// TwinCAT 3 PLC project mobject_graph_plc_pack
// Title: mobject-graph-plc-pack
// Company: mobject
// Author: mobject dev team
// ProjectVersion: 0.19.0
// ProgramVersion: 3.1.4026.22
// libraries:
//   mobject-core,0.10.0,mobject
//   mobject-graph,0.18.0,mobject
//   Tc2_Standard, * (Beckhoff Automation GmbH)
//   Tc2_System, * (Beckhoff Automation GmbH)
//   Tc2_Utilities, * (Beckhoff Automation GmbH)
//   Tc3_Module, * (Beckhoff Automation GmbH)
// project tree:
//   Datatypes/Arrays/ _Array0To7OfByte.TcPOU (not stored)
//   Datatypes/ PlcDatatypePack.TcPOU
//   Datatypes/Structs/ _GUID.TcPOU, _TIMESTRUCT.TcPOU (not stored)
//   Nodes/Converter/DINT_TO_/ Node_DINT_TO_LREAL.TcPOU, Node_DINT_TO_REAL.TcPOU
//   Nodes/Converter/LREAL_TO_/ Node_LREAL_TO_UDINT.TcPOU, Node_LREAL_TO_DINT.TcPOU
//   Nodes/Converter/REAL_TO_/ Node_REAL_TO_UDINT.TcPOU, Node_REAL_TO_DINT.TcPOU
//   Nodes/Converter/UDINT_TO_/ Node_UDINT_TO_REAL.TcPOU, Node_UDINT_TO_LREAL.TcPOU
//   Nodes/Flow/ Node_ForNext.TcPOU, Node_IF.TcPOU, Node_IF_Merge.TcPOU
//   Nodes/Hardware/Digital/ Node_DigitalInput.TcPOU, Node_DigitalOutput.TcPOU
//   Nodes/Logic/ Node_OR.TcPOU, Node_NOT.TcPOU, Node_AND.TcPOU, Node_NOR.TcPOU, Node_NAND.TcPOU, Node_XOR.TcPOU, Node_XNOR.TcPOU
//   Nodes/ PlcNodePack.TcPOU
//   Datatypes/Alias/ _FLOAT.TcPOU (not stored), _HRESULT.TcPOU (not stored)
//   Datatypes/Enums/ _E_TcEventClass.TcPOU (not stored)
//   Nodes/Strings/ Node_CONCAT.TcPOU, Node_DELETE.TcPOU, Node_REPLACE.TcPOU, Node_MID.TcPOU, Node_INSERT.TcPOU, Node_FIND.TcPOU, Node_LEFT.TcPOU, Node_RIGHT.TcPOU, Node_LEN.TcPOU
//   Nodes/TwinCAT/ Node_TwinCATStatus.TcPOU
//   Nodes/Variable/ Node_SetByRef.TcPOU
//   / PlcPack.TcPOU

// ---- Datatypes/PlcDatatypePack.TcPOU
{attribute 'linkalways'} 
{attribute 'no_explicit_call' := 'This FB is a CLASS and must be accessed using methods or properties'}
{attribute 'enable_dynamic_creation'}
FUNCTION_BLOCK PlcDatatypePack
VAR
	
	// alias
    _float : _FLOAT(0.0);
	_hresult : _HRESULT(0);

	// enums
	_e_TcEventClass : _E_TcEventClass(E_TcEventClass.TCEVENTCLASS_NONE);
	
	// structures
	_timestruct : _TIMESTRUCT();
	
END_VAR

METHOD RegisterWithDatatypes
VAR_INPUT
	Datatypes : I_Datatypes;
END_VAR
// alias
Datatypes.RegisterDatatype(_float);
Datatypes.RegisterDatatype(_hresult);

// enums
Datatypes.RegisterDatatype(_e_TcEventClass);

// structures
Datatypes.RegisterDatatype(_timestruct);
END_METHOD

END_FUNCTION_BLOCK

// ---- Datatypes/Structs/_GUID.TcPOU
{attribute 'linkalways'} 
{attribute 'no_explicit_call' := 'This FB is a CLASS and must be accessed using methods or properties'}
{attribute 'enable_dynamic_creation'}
FUNCTION_BLOCK _GUID EXTENDS StructuredDatatypeBase
VAR
	localData : GUID;
	activeData : REFERENCE TO GUID REF= localData;
	_data1 : _DWORD(localData.data1);
	_data2 : _WORD(localData.data2);
    _data3 : _WORD(localData.data3);
	_data4 : _Array0To7OfByte();
END_VAR

PROPERTY PUBLIC Address : PVOID
GET
Address := ADR(activeData);
END_GET
END_PROPERTY

METHOD PUBLIC ClearReference
VAR_INPUT
END_VAR
activeData REF= localData;
SetMemberReference();
END_METHOD

METHOD PUBLIC Clone : I_Datatype
VAR
    pClone : POINTER TO _GUID;
END_VAR
pClone := __NEW(_GUID());
pClone^.Value := Value;
Clone := pClone^;
END_METHOD

PROPERTY PUBLIC Data1 : REFERENCE TO _DWORD
GET
Data1 REF= _data1;
END_GET
END_PROPERTY

PROPERTY PUBLIC Data2 : REFERENCE TO _WORD
GET
Data2 REF= _data2;
END_GET
END_PROPERTY

PROPERTY PUBLIC Data3 : REFERENCE TO _WORD
GET
Data3 REF= _data3;
END_GET
END_PROPERTY

PROPERTY PUBLIC Data4 : REFERENCE TO _Array0To7OfByte
GET
Data4 REF= _data4;
END_GET
END_PROPERTY

METHOD PUBLIC EqualsGuid : BOOL
VAR_INPUT
	guid : GUID;
END_VAR
EqualsGuid := GuidsEqual(adr(guid), this^.Address);
END_METHOD

METHOD FB_init : BOOL
VAR_INPUT
	bInitRetains : BOOL; // if TRUE, the retain variables are initialized (warm start / cold start)
	bInCopyCode : BOOL;  // if TRUE, the instance afterwards gets moved into the copy code (online change)
END_VAR
SetMemberReference();
AddMember('Data1',_data1);
AddMember('Data2',_data2);
AddMember('Data3',_data3);
AddMember('Data4',_data4);
END_METHOD

PROPERTY PUBLIC Identifier : T_MAXSTRING
GET
Identifier := 'GUID';
END_GET
END_PROPERTY

METHOD PROTECTED IsValidGuidString : BOOL
VAR_INPUT
	GuidAsString : STRING;
END_VAR
VAR
	position : INT;
	stringIndex : INT;
	dashCount : INT := 0;
END_VAR
VAR CONSTANT
	CHARACTER_HYPHEN : BYTE := 16#2D;
	CHARACTER_0 : BYTE := 16#30;
	CHARACTER_9 : BYTE := 16#39;
	CHARACTER_A : BYTE := 16#41;
	CHARACTER_F : BYTE := 16#46;
	CHARACTER_LCASE_A : BYTE := 16#61;
	CHARACTER_LCASE_F : BYTE := 16#66;
END_VAR
// Check the overall length of the string (36 including 4 dashes)
IF LEN(GuidAsString) <> 36 THEN
	RETURN;
END_IF

// Check each character
FOR position := 1 TO 36 DO
	stringIndex := position - 1; 
	CASE position OF
		9, 14, 19, 24:
			// Dashes should be at positions 9, 14, 19, 24
			IF GuidAsString[stringIndex] <> CHARACTER_HYPHEN THEN
				RETURN;
			ELSE
				dashCount := dashCount + 1;
			END_IF
		ELSE
			// All other positions should contain hex digits (0-9, A-F, a-f)
			IF NOT ((GuidAsString[stringIndex] >= CHARACTER_0 AND GuidAsString[stringIndex] <= CHARACTER_9) OR 
				(GuidAsString[stringIndex] >= CHARACTER_A AND GuidAsString[stringIndex] <= CHARACTER_F) OR 
				(GuidAsString[stringIndex] >= CHARACTER_LCASE_A AND GuidAsString[stringIndex] <= CHARACTER_LCASE_F)) THEN
				RETURN;
			END_IF
	END_CASE
END_FOR

// Ensure exactly four dashes are present
IF dashCount = 4 THEN
	IsValidGuidString := TRUE;
END_IF
END_METHOD

METHOD PUBLIC MakeReferenceTo
VAR_INPUT
	ReferenceTarget : REFERENCE TO GUID;
END_VAR
activeData REF= ReferenceTarget;
SetMemberReference();
END_METHOD

METHOD PROTECTED SetMemberReference
VAR_INPUT
END_VAR
_data1.MakeReferenceTo(activeData.Data1);
_data2.MakeReferenceTo(activeData.Data2);
_data3.MakeReferenceTo(activeData.Data3);
_data4.MakeReferenceTo(activeData.Data4);
END_METHOD

PROPERTY PUBLIC Size : UDINT
GET
Size := SIZEOF(activeData);
END_GET
END_PROPERTY

METHOD PUBLIC ToString : T_MAXSTRING
VAR_INPUT
END_VAR
ToString := GUID_TO_STRING(activeData);
END_METHOD

METHOD TryDeserializeFrom : BOOL
VAR_INPUT
	Deserializer : I_Deserializer;
	Feedback : I_DeserializerFeedback;
END_VAR
VAR
	localFeedback : DeserializerFeedback;
	guidAsString : T_MAXSTRING;
END_VAR
// this customized version of TryDeserializeFrom allows for the use of string guids. 
// if a string is not found, then it will try to deserialize from an object.
IF Deserializer.TryGetString(guidAsString, localFeedback) THEN	
	IF TryFromString(guidAsString) THEN
		TryDeserializeFrom := TRUE;
		RETURN;
	END_IF
	
	Feedback.LogDeserializationFailedError('Invalid GUID String');	
	RETURN;
END_IF

TryDeserializeFrom := SUPER^.TryDeserializeFrom(Deserializer, Feedback);
END_METHOD

METHOD PUBLIC TryFromString : BOOL;
VAR_INPUT
	GuidAsString : T_MAXSTRING;
END_VAR
IF NOT IsValidGuidString(GuidAsString) THEN
	RETURN;
END_IF

activeData := STRING_TO_GUID(GuidAsString);
TryFromString := true;
END_METHOD

METHOD TryMakeReferenceTo : BOOL
VAR_INPUT
	Target : I_Datatype;
END_VAR
VAR
	pTargetData : POINTER TO GUID;
END_VAR
IF NOT IsEquivalentTo(Target) THEN
	RETURN;
END_IF

pTargetData := Target.Address;
activeData REF= pTargetData^;
SetMemberReference();
TryMakeReferenceTo := TRUE;
END_METHOD

PROPERTY PUBLIC Value : REFERENCE TO GUID
GET
Value REF= activeData;
END_GET
END_PROPERTY

END_FUNCTION_BLOCK

// ---- Nodes/Converter/DINT_TO_/Node_DINT_TO_LREAL.TcPOU
{attribute 'linkalways'} 
{attribute 'no_explicit_call' := 'This FB is a CLASS and must be accessed using methods or properties'}
{attribute 'enable_dynamic_creation'}
FUNCTION_BLOCK FINAL Node_DINT_TO_LREAL EXTENDS Node
VAR
	in : _DINT(0);
	out : _LREAL(0.0);
	success : _BOOL(FALSE);
END_VAR

METHOD PUBLIC  Clone : I_Node
VAR
	pNode : POINTER TO Node_DINT_TO_LREAL;
END_VAR
pNode := __NEW(Node_DINT_TO_LREAL);
Clone := pNode^;
END_METHOD

METHOD FB_init : BOOL
VAR_INPUT
	bInitRetains : BOOL; // if TRUE, the retain variables are initialized (warm start / cold start)
	bInCopyCode : BOOL;  // if TRUE, the instance afterwards gets moved into the copy code (online change)
END_VAR
AddParameter('in', in);
AddOutput('out', out);
AddOutput('success', success);

this^.Metadatum.AddBoolAsMetadata('deprecated', true);
END_METHOD

METHOD PROTECTED OnExecute
VAR
END_VAR
success.Value := TryConvert_DINT_TO_LREAL(in.Value, out.Value);
END_METHOD

END_FUNCTION_BLOCK

// ---- Nodes/Converter/DINT_TO_/Node_DINT_TO_REAL.TcPOU
{attribute 'linkalways'} 
{attribute 'no_explicit_call' := 'This FB is a CLASS and must be accessed using methods or properties'}
{attribute 'enable_dynamic_creation'}
FUNCTION_BLOCK FINAL Node_DINT_TO_REAL EXTENDS Node
VAR
	in : _DINT(0);
	out : _REAL(0.0);
	success : _BOOL(FALSE);
END_VAR

METHOD PUBLIC  Clone : I_Node
VAR
	pNode : POINTER TO Node_DINT_TO_REAL;
END_VAR
pNode := __NEW(Node_DINT_TO_REAL);
Clone := pNode^;
END_METHOD

METHOD FB_init : BOOL
VAR_INPUT
	bInitRetains : BOOL; // if TRUE, the retain variables are initialized (warm start / cold start)
	bInCopyCode : BOOL;  // if TRUE, the instance afterwards gets moved into the copy code (online change)
END_VAR
AddParameter('in', in);
AddOutput('out', out);
AddOutput('success', success);

this^.Metadatum.AddBoolAsMetadata('deprecated', true);
END_METHOD

METHOD PROTECTED OnExecute
VAR
END_VAR
success.Value := TryConvert_DINT_TO_REAL(in.Value, out.Value);
END_METHOD

END_FUNCTION_BLOCK

// ---- Nodes/Converter/LREAL_TO_/Node_LREAL_TO_UDINT.TcPOU
{attribute 'linkalways'} 
{attribute 'no_explicit_call' := 'This FB is a CLASS and must be accessed using methods or properties'}
{attribute 'enable_dynamic_creation'}
FUNCTION_BLOCK FINAL Node_LREAL_TO_UDINT EXTENDS Node
VAR
	in : _LREAL(0.0);
	out : _UDINT(0);
	success : _BOOL(FALSE);
END_VAR

METHOD PUBLIC  Clone : I_Node
VAR
	pNode : POINTER TO Node_LREAL_TO_UDINT;
END_VAR
pNode := __NEW(Node_LREAL_TO_UDINT);
Clone := pNode^;
END_METHOD

METHOD FB_init : BOOL
VAR_INPUT
	bInitRetains : BOOL; // if TRUE, the retain variables are initialized (warm start / cold start)
	bInCopyCode : BOOL;  // if TRUE, the instance afterwards gets moved into the copy code (online change)
END_VAR
AddParameter('in', in);
AddOutput('out', out);
AddOutput('success', success);

this^.Metadatum.AddBoolAsMetadata('deprecated', true);
END_METHOD

METHOD PROTECTED OnExecute
VAR
END_VAR
success.Value := TryConvert_LREAL_TO_UDINT(in.Value, out.Value);
END_METHOD

END_FUNCTION_BLOCK

// ---- Nodes/Converter/LREAL_TO_/Node_LREAL_TO_DINT.TcPOU
{attribute 'linkalways'} 
{attribute 'no_explicit_call' := 'This FB is a CLASS and must be accessed using methods or properties'}
{attribute 'enable_dynamic_creation'}
FUNCTION_BLOCK FINAL Node_LREAL_TO_DINT EXTENDS Node
VAR
	in : _LREAL(0.0);
	out : _DINT(0);
	success : _BOOL(FALSE);
END_VAR

METHOD PUBLIC  Clone : I_Node
VAR
	pNode : POINTER TO Node_LREAL_TO_DINT;
END_VAR
pNode := __NEW(Node_LREAL_TO_DINT);
Clone := pNode^;
END_METHOD

METHOD FB_init : BOOL
VAR_INPUT
	bInitRetains : BOOL; // if TRUE, the retain variables are initialized (warm start / cold start)
	bInCopyCode : BOOL;  // if TRUE, the instance afterwards gets moved into the copy code (online change)
END_VAR
AddParameter('in', in);
AddOutput('out', out);
AddOutput('success', success);

this^.Metadatum.AddBoolAsMetadata('deprecated', true);
END_METHOD

METHOD PROTECTED OnExecute
VAR
END_VAR
success.Value := TryConvert_LREAL_TO_DINT(in.Value, out.Value);
END_METHOD

END_FUNCTION_BLOCK

// ---- Nodes/Converter/REAL_TO_/Node_REAL_TO_UDINT.TcPOU
{attribute 'linkalways'} 
{attribute 'no_explicit_call' := 'This FB is a CLASS and must be accessed using methods or properties'}
{attribute 'enable_dynamic_creation'}
FUNCTION_BLOCK FINAL Node_REAL_TO_UDINT EXTENDS Node
VAR
	in : _REAL(0.0);
	out : _UDINT(0);
	success : _BOOL(FALSE);
END_VAR

METHOD PUBLIC  Clone : I_Node
VAR
	pNode : POINTER TO Node_REAL_TO_UDINT;
END_VAR
pNode := __NEW(Node_REAL_TO_UDINT);
Clone := pNode^;
END_METHOD

METHOD FB_init : BOOL
VAR_INPUT
	bInitRetains : BOOL; // if TRUE, the retain variables are initialized (warm start / cold start)
	bInCopyCode : BOOL;  // if TRUE, the instance afterwards gets moved into the copy code (online change)
END_VAR
AddParameter('in', in);
AddOutput('out', out);
AddOutput('success', success);

this^.Metadatum.AddBoolAsMetadata('deprecated', true);
END_METHOD

METHOD PROTECTED OnExecute
VAR
END_VAR
success.Value := TryConvert_REAL_TO_UDINT(in.Value, out.Value);
END_METHOD

END_FUNCTION_BLOCK

// ---- Nodes/Converter/REAL_TO_/Node_REAL_TO_DINT.TcPOU
{attribute 'linkalways'} 
{attribute 'no_explicit_call' := 'This FB is a CLASS and must be accessed using methods or properties'}
{attribute 'enable_dynamic_creation'}
FUNCTION_BLOCK FINAL Node_REAL_TO_DINT EXTENDS Node
VAR
	in : _REAL(0.0);
	out : _DINT(0);
	success : _BOOL(FALSE);
END_VAR

METHOD PUBLIC  Clone : I_Node
VAR
	pNode : POINTER TO Node_REAL_TO_DINT;
END_VAR
pNode := __NEW(Node_REAL_TO_DINT);
Clone := pNode^;
END_METHOD

METHOD FB_init : BOOL
VAR_INPUT
	bInitRetains : BOOL; // if TRUE, the retain variables are initialized (warm start / cold start)
	bInCopyCode : BOOL;  // if TRUE, the instance afterwards gets moved into the copy code (online change)
END_VAR
AddParameter('in', in);
AddOutput('out', out);
AddOutput('success', success);

this^.Metadatum.AddBoolAsMetadata('deprecated', true);
END_METHOD

METHOD PROTECTED OnExecute
VAR
END_VAR
success.Value := TryConvert_REAL_TO_DINT(in.Value, out.Value);
END_METHOD

END_FUNCTION_BLOCK

// ---- Nodes/Converter/UDINT_TO_/Node_UDINT_TO_REAL.TcPOU
{attribute 'linkalways'} 
{attribute 'no_explicit_call' := 'This FB is a CLASS and must be accessed using methods or properties'}
{attribute 'enable_dynamic_creation'}
FUNCTION_BLOCK FINAL Node_UDINT_TO_REAL EXTENDS Node
VAR
	in : _UDINT(0);
	out : _REAL(0.0);
	success : _BOOL(FALSE);
END_VAR

METHOD PUBLIC  Clone : I_Node
VAR
	pNode : POINTER TO Node_UDINT_TO_REAL;
END_VAR
pNode := __NEW(Node_UDINT_TO_REAL);
Clone := pNode^;
END_METHOD

METHOD FB_init : BOOL
VAR_INPUT
	bInitRetains : BOOL; // if TRUE, the retain variables are initialized (warm start / cold start)
	bInCopyCode : BOOL;  // if TRUE, the instance afterwards gets moved into the copy code (online change)
END_VAR
AddParameter('in', in);
AddOutput('out', out);
AddOutput('success', success);

this^.Metadatum.AddBoolAsMetadata('deprecated', true);
END_METHOD

METHOD PROTECTED OnExecute
VAR
END_VAR
success.Value := TryConvert_UDINT_TO_REAL(in.Value, out.Value);
END_METHOD

END_FUNCTION_BLOCK

// ---- Nodes/Converter/UDINT_TO_/Node_UDINT_TO_LREAL.TcPOU
{attribute 'linkalways'} 
{attribute 'no_explicit_call' := 'This FB is a CLASS and must be accessed using methods or properties'}
{attribute 'enable_dynamic_creation'}
FUNCTION_BLOCK FINAL Node_UDINT_TO_LREAL EXTENDS Node
VAR
	in : _UDINT(0);
	out : _LREAL(0.0);
	success : _BOOL(FALSE);
END_VAR

METHOD PUBLIC  Clone : I_Node
VAR
	pNode : POINTER TO Node_UDINT_TO_LREAL;
END_VAR
pNode := __NEW(Node_UDINT_TO_LREAL);
Clone := pNode^;
END_METHOD

METHOD FB_init : BOOL
VAR_INPUT
	bInitRetains : BOOL; // if TRUE, the retain variables are initialized (warm start / cold start)
	bInCopyCode : BOOL;  // if TRUE, the instance afterwards gets moved into the copy code (online change)
END_VAR
AddParameter('in', in);
AddOutput('out', out);
AddOutput('success', success);

this^.Metadatum.AddBoolAsMetadata('deprecated', true);
END_METHOD

METHOD PROTECTED OnExecute
VAR
END_VAR
success.Value := TryConvert_UDINT_TO_LREAL(in.Value, out.Value);
END_METHOD

END_FUNCTION_BLOCK

// ---- Nodes/Flow/Node_ForNext.TcPOU
{attribute 'linkalways'} 
{attribute 'no_explicit_call' := 'This FB is a CLASS and must be accessed using methods or properties'}
{attribute 'enable_dynamic_creation'}
FUNCTION_BLOCK Node_ForNext EXTENDS Node
VAR
	startValue : _DINT(0);
	endValue : _DINT(1);
	step : _DINT(1);	
	doEvent : I_EventOutputPort := AddEventOutput('do');
	index : _DINT(0);
END_VAR

METHOD PUBLIC  Clone : I_Node
VAR_INPUT
END_VAR
VAR
	pNode : POINTER TO Node_ForNext;
END_VAR
pNode := __NEW(Node_ForNext);
Clone := pNode^;
END_METHOD

METHOD FB_init : BOOL
VAR_INPUT
	bInitRetains : BOOL; // if TRUE, the retain variables are initialized (warm start / cold start)
	bInCopyCode : BOOL;  // if TRUE, the instance afterwards gets moved into the copy code (online change)
END_VAR
AddParameter('start', startValue);
AddParameter('end', endValue);
AddParameter('step', step);
AddOutput('index', index);

THIS^.Metadatum.AddBoolAsMetadata('development', TRUE);
END_METHOD

METHOD PROTECTED  OnExecute
VAR
	i : DINT;
END_VAR
FOR i := startValue.Value TO endValue.Value BY step.Value DO
	index.Value := i;
	doEvent.Trigger();
END_FOR
END_METHOD

END_FUNCTION_BLOCK

// ---- Nodes/Flow/Node_IF.TcPOU
{attribute 'linkalways'} 
{attribute 'no_explicit_call' := 'This FB is a CLASS and must be accessed using methods or properties'}
{attribute 'enable_dynamic_creation'}
FUNCTION_BLOCK Node_IF EXTENDS Node
VAR
	condition : _BOOL(FALSE);
	isTrue : I_EventOutputPort := AddEventOutput('isTrue');
	isFalse : I_EventOutputPort := AddEventOutput('isFalse');
END_VAR

METHOD PUBLIC  Clone : I_Node
VAR_INPUT
END_VAR
VAR
	pNode : POINTER TO Node_IF;
END_VAR
pNode := __NEW(Node_IF);
Clone := pNode^;
END_METHOD

METHOD FB_init : BOOL
VAR_INPUT
	bInitRetains : BOOL; // if TRUE, the retain variables are initialized (warm start / cold start)
	bInCopyCode : BOOL;  // if TRUE, the instance afterwards gets moved into the copy code (online change)
END_VAR
AddInput('condition', condition);

THIS^.Metadatum.AddBoolAsMetadata('development', TRUE);
END_METHOD

METHOD PROTECTED  OnExecute
IF condition.Value THEN
	isTrue.Trigger();
ELSE
	isFalse.Trigger();
END_IF
END_METHOD

END_FUNCTION_BLOCK

// ---- Nodes/Flow/Node_IF_Merge.TcPOU
{attribute 'linkalways'} 
{attribute 'no_explicit_call' := 'This FB is a CLASS and must be accessed using methods or properties'}
{attribute 'enable_dynamic_creation'}
FUNCTION_BLOCK Node_IF_Merge EXTENDS Node
VAR
	selectA : TriggerWatchEventPortAction();
	selectB : TriggerWatchEventPortAction();
	a : _ANY();
	b : _ANY();
	out  : _ANY();
END_VAR

METHOD PUBLIC  Clone : I_Node
VAR_INPUT
END_VAR
VAR
	pNode : POINTER TO Node_IF_Merge;
END_VAR
pNode := __NEW(Node_IF_Merge);
Clone := pNode^;
END_METHOD

METHOD FB_init : BOOL
VAR_INPUT
	bInitRetains : BOOL; // if TRUE, the retain variables are initialized (warm start / cold start)
	bInCopyCode : BOOL;  // if TRUE, the instance afterwards gets moved into the copy code (online change)
END_VAR
AddEventInput('selectA', selectA);
AddEventInput('selectB', selectB);
AddInputWithGroup('a',a,'T');
AddInputWithGroup('b',b,'T');
AddOutputWithGroup('out',out,'T');

THIS^.Metadatum.AddBoolAsMetadata('development', TRUE);
END_METHOD

METHOD PROTECTED  OnExecute
IF selectA.WasTriggered THEN
	out.TryCopyFrom(a);
END_IF

IF selectB.WasTriggered THEN
	out.TryCopyFrom(b);
END_IF

selectA.ResetWatch();
selectB.ResetWatch();
END_METHOD

END_FUNCTION_BLOCK

// ---- Nodes/Hardware/Digital/Node_DigitalInput.TcPOU
{attribute 'linkalways'} 
{attribute 'no_explicit_call' := 'This FB is a CLASS and must be accessed using methods or properties'}
{attribute 'enable_dynamic_creation'}
FUNCTION_BLOCK FINAL Node_DigitalInput EXTENDS HardwareNode
VAR
	input AT %I* : BOOL;
	out : _BOOL(FALSE);
END_VAR

METHOD FB_init : BOOL
VAR_INPUT
	bInitRetains : BOOL; // if TRUE, the retain variables are initialized (warm start / cold start)
	bInCopyCode : BOOL;  // if TRUE, the instance afterwards gets moved into the copy code (online change)
END_VAR
AddOutput('out', out);
END_METHOD

METHOD PROTECTED OnExecute
VAR
END_VAR
out.Value := input;
END_METHOD

END_FUNCTION_BLOCK

// ---- Nodes/Hardware/Digital/Node_DigitalOutput.TcPOU
{attribute 'linkalways'} 
{attribute 'no_explicit_call' := 'This FB is a CLASS and must be accessed using methods or properties'}
{attribute 'enable_dynamic_creation'}
FUNCTION_BLOCK FINAL Node_DigitalOutput EXTENDS HardwareNode
VAR
	output AT %Q* : BOOL;
	in : _BOOL(FALSE);
END_VAR

METHOD FB_init : BOOL
VAR_INPUT
	bInitRetains : BOOL; // if TRUE, the retain variables are initialized (warm start / cold start)
	bInCopyCode : BOOL;  // if TRUE, the instance afterwards gets moved into the copy code (online change)
END_VAR
AddParameter('in', in);
END_METHOD

METHOD PROTECTED OnExecute
VAR
END_VAR
output := in.Value;
END_METHOD

END_FUNCTION_BLOCK

// ---- Nodes/Logic/Node_OR.TcPOU
{attribute 'linkalways'} 
{attribute 'no_explicit_call' := 'This FB is a CLASS and must be accessed using methods or properties'}
{attribute 'enable_dynamic_creation'}
FUNCTION_BLOCK FINAL Node_OR EXTENDS Node
VAR
	in1 : _BOOL(FALSE);
    in2 : _BOOL(FALSE);
	out : _BOOL(FALSE);
END_VAR

METHOD PUBLIC  Clone : I_Node
VAR
	pNode : POINTER TO Node_OR;
END_VAR
pNode := __NEW(Node_OR);
Clone := pNode^;
END_METHOD

METHOD FB_init : BOOL
VAR_INPUT
	bInitRetains : BOOL; // if TRUE, the retain variables are initialized (warm start / cold start)
	bInCopyCode : BOOL;  // if TRUE, the instance afterwards gets moved into the copy code (online change)
END_VAR
AddParameter('in1', in1);
AddParameter('in2', in2);
AddOutput('out', out);

this^.Metadatum.AddBoolAsMetadata('deprecated', true);
END_METHOD

METHOD PROTECTED OnExecute
VAR
END_VAR
out.Value := in1.Value OR in2.Value;
END_METHOD

END_FUNCTION_BLOCK

// ---- Nodes/Logic/Node_NOT.TcPOU
{attribute 'linkalways'} 
{attribute 'no_explicit_call' := 'This FB is a CLASS and must be accessed using methods or properties'}
{attribute 'enable_dynamic_creation'}
FUNCTION_BLOCK FINAL Node_NOT EXTENDS Node
VAR
	in : _BOOL(FALSE);
	out : _BOOL(FALSE);
END_VAR

METHOD PUBLIC  Clone : I_Node
VAR
	pNode : POINTER TO Node_NOT;
END_VAR
pNode := __NEW(Node_NOT);
Clone := pNode^;
END_METHOD

METHOD FB_init : BOOL
VAR_INPUT
	bInitRetains : BOOL; // if TRUE, the retain variables are initialized (warm start / cold start)
	bInCopyCode : BOOL;  // if TRUE, the instance afterwards gets moved into the copy code (online change)
END_VAR
AddParameter('in', in);
AddOutput('out', out);

this^.Metadatum.AddBoolAsMetadata('deprecated', true);
END_METHOD

METHOD PROTECTED OnExecute
VAR
END_VAR
out.Value := NOT in.Value;
END_METHOD

END_FUNCTION_BLOCK

// ---- Nodes/Logic/Node_AND.TcPOU
{attribute 'linkalways'} 
{attribute 'no_explicit_call' := 'This FB is a CLASS and must be accessed using methods or properties'}
{attribute 'enable_dynamic_creation'}
FUNCTION_BLOCK FINAL Node_AND EXTENDS Node
VAR
	in1 : _BOOL(FALSE);
    in2 : _BOOL(FALSE);
	out : _BOOL(FALSE);
END_VAR

METHOD PUBLIC  Clone : I_Node
VAR
	pNode : POINTER TO Node_AND;
END_VAR
pNode := __NEW(Node_AND);
Clone := pNode^;
END_METHOD

METHOD FB_init : BOOL
VAR_INPUT
	bInitRetains : BOOL; // if TRUE, the retain variables are initialized (warm start / cold start)
	bInCopyCode : BOOL;  // if TRUE, the instance afterwards gets moved into the copy code (online change)
END_VAR
AddParameter('in1', in1);
AddParameter('in2', in2);
AddOutput('out', out);
END_METHOD

METHOD PROTECTED OnExecute
VAR
END_VAR
out.Value := in1.Value AND in2.Value;
END_METHOD

END_FUNCTION_BLOCK

// ---- Nodes/Logic/Node_NOR.TcPOU
{attribute 'linkalways'} 
{attribute 'no_explicit_call' := 'This FB is a CLASS and must be accessed using methods or properties'}
{attribute 'enable_dynamic_creation'}
FUNCTION_BLOCK FINAL Node_NOR EXTENDS Node
VAR
	in1 : _BOOL(FALSE);
    in2 : _BOOL(FALSE);
	out : _BOOL(FALSE);
END_VAR

METHOD PUBLIC  Clone : I_Node
VAR
	pNode : POINTER TO Node_NOR;
END_VAR
pNode := __NEW(Node_NOR);
Clone := pNode^;
END_METHOD

METHOD FB_init : BOOL
VAR_INPUT
	bInitRetains : BOOL; // if TRUE, the retain variables are initialized (warm start / cold start)
	bInCopyCode : BOOL;  // if TRUE, the instance afterwards gets moved into the copy code (online change)
END_VAR
AddParameter('in1', in1);
AddParameter('in2', in2);
AddOutput('out', out);

this^.Metadatum.AddBoolAsMetadata('deprecated', true);
END_METHOD

METHOD PROTECTED OnExecute
VAR
END_VAR
out.Value := NOT(in1.Value OR in2.Value);
END_METHOD

END_FUNCTION_BLOCK

// ---- Nodes/Logic/Node_NAND.TcPOU
{attribute 'linkalways'} 
{attribute 'no_explicit_call' := 'This FB is a CLASS and must be accessed using methods or properties'}
{attribute 'enable_dynamic_creation'}
FUNCTION_BLOCK FINAL Node_NAND EXTENDS Node
VAR
	in1 : _BOOL(FALSE);
    in2 : _BOOL(FALSE);
	out : _BOOL(FALSE);
END_VAR

METHOD PUBLIC  Clone : I_Node
VAR
	pNode : POINTER TO Node_NAND;
END_VAR
pNode := __NEW(Node_NAND);
Clone := pNode^;
END_METHOD

METHOD FB_init : BOOL
VAR_INPUT
	bInitRetains : BOOL; // if TRUE, the retain variables are initialized (warm start / cold start)
	bInCopyCode : BOOL;  // if TRUE, the instance afterwards gets moved into the copy code (online change)
END_VAR
AddParameter('in1', in1);
AddParameter('in2', in2);
AddOutput('out', out);

this^.Metadatum.AddBoolAsMetadata('deprecated', true);
END_METHOD

METHOD PROTECTED OnExecute
VAR
END_VAR
out.Value := NOT(in1.Value AND in2.Value);
END_METHOD

END_FUNCTION_BLOCK

// ---- Nodes/Logic/Node_XOR.TcPOU
{attribute 'linkalways'} 
{attribute 'no_explicit_call' := 'This FB is a CLASS and must be accessed using methods or properties'}
{attribute 'enable_dynamic_creation'}
FUNCTION_BLOCK FINAL Node_XOR EXTENDS Node
VAR
	in1 : _BOOL(FALSE);
    in2 : _BOOL(FALSE);
	out : _BOOL(FALSE);
END_VAR

METHOD PUBLIC  Clone : I_Node
VAR
	pNode : POINTER TO Node_XOR;
END_VAR
pNode := __NEW(Node_XOR);
Clone := pNode^;
END_METHOD

METHOD FB_init : BOOL
VAR_INPUT
	bInitRetains : BOOL; // if TRUE, the retain variables are initialized (warm start / cold start)
	bInCopyCode : BOOL;  // if TRUE, the instance afterwards gets moved into the copy code (online change)
END_VAR
AddParameter('in1', in1);
AddParameter('in2', in2);
AddOutput('out', out);

this^.Metadatum.AddBoolAsMetadata('deprecated', true);
END_METHOD

METHOD PROTECTED OnExecute
VAR
END_VAR
out.Value := in1.Value XOR in2.Value;
END_METHOD

END_FUNCTION_BLOCK

// ---- Nodes/Logic/Node_XNOR.TcPOU
{attribute 'linkalways'} 
{attribute 'no_explicit_call' := 'This FB is a CLASS and must be accessed using methods or properties'}
{attribute 'enable_dynamic_creation'}
FUNCTION_BLOCK FINAL Node_XNOR EXTENDS Node
VAR
	in1 : _BOOL(FALSE);
    in2 : _BOOL(FALSE);
	out : _BOOL(FALSE);
END_VAR

METHOD PUBLIC  Clone : I_Node
VAR
	pNode : POINTER TO Node_XNOR;
END_VAR
pNode := __NEW(Node_XNOR);
Clone := pNode^;
END_METHOD

METHOD FB_init : BOOL
VAR_INPUT
	bInitRetains : BOOL; // if TRUE, the retain variables are initialized (warm start / cold start)
	bInCopyCode : BOOL;  // if TRUE, the instance afterwards gets moved into the copy code (online change)
END_VAR
AddParameter('in1', in1);
AddParameter('in2', in2);
AddOutput('out', out);

this^.Metadatum.AddBoolAsMetadata('deprecated', true);
END_METHOD

METHOD PROTECTED OnExecute
VAR
END_VAR
out.Value := NOT(in1.Value XOR in2.Value);
END_METHOD

END_FUNCTION_BLOCK

// ---- Nodes/PlcNodePack.TcPOU
{attribute 'linkalways'} 
{attribute 'no_explicit_call' := 'This FB is a CLASS and must be accessed using methods or properties'}
{attribute 'enable_dynamic_creation'}
FUNCTION_BLOCK PlcNodePack
VAR
    // Conversion
	// DINT_TO
	node_DINT_TO_LREAL : Node_DINT_TO_LREAL;
	node_DINT_TO_REAL : Node_DINT_TO_REAL;
	// LREAL_TO_
	node_LREAL_TO_DINT : Node_LREAL_TO_DINT;
	node_LREAL_TO_UDINT : Node_LREAL_TO_UDINT;
	// REAL_TO_
    node_REAL_TO_DINT : Node_REAL_TO_DINT;
	node_REAL_TO_UDINT : Node_REAL_TO_UDINT;
	// UDINT_TO
	node_UDINT_TO_LREAL : Node_UDINT_TO_LREAL;
	node_UDINT_TO_REAL : Node_UDINT_TO_REAL;
    // Logic
    node_NOT : Node_NOT;
    node_AND : Node_AND;
    node_NAND : Node_NAND;
    node_OR : Node_OR;
    node_NOR : Node_NOR;
    node_XOR : Node_XOR;
    node_XNOR : Node_XNOR;
	
	// Flow
	nodeIf : Node_If;
	nodeIfMerge : Node_if_merge;
	nodeForNext : Node_ForNext;
	
	// TwinCAT
	node_TwinCATStatus : Node_TwinCATStatus;
	
	// Strings
	node_CONCAT : Node_CONCAT;
    node_DELETE : Node_DELETE;
    node_FIND : Node_FIND;
    node_INSERT : Node_INSERT;
    node_LEFT : Node_LEFT;
    node_LEN : Node_LEN;
    node_MID : Node_MID;
	node_REPLACE : Node_REPLACE;
    node_RIGHT : Node_RIGHT;
	
	// variable
	node_SetByRef : Node_SetByRef;
	
END_VAR

METHOD PUBLIC RegisterWithNodeFactory
VAR_INPUT
	NodeFactory : I_NodeFactory;
END_VAR
// Conversion
NodeFactory.AddNodeAsPrototype('PLC/Convert/DINT/DINT_TO_LREAL', node_DINT_TO_LREAL);
NodeFactory.AddNodeAsPrototype('PLC/Convert/DINT/DINT_TO_REAL', node_DINT_TO_REAL);
NodeFactory.AddNodeAsPrototype('PLC/Convert/LREAL/LREAL_TO_DINT', node_LREAL_TO_DINT);
NodeFactory.AddNodeAsPrototype('PLC/Convert/LREAL/LREAL_TO_UDINT', node_LREAL_TO_UDINT);
NodeFactory.AddNodeAsPrototype('PLC/Convert/REAL/REAL_TO_DINT', node_REAL_TO_DINT);
NodeFactory.AddNodeAsPrototype('PLC/Convert/REAL/REAL_TO_UDINT', node_REAL_TO_UDINT);
NodeFactory.AddNodeAsPrototype('PLC/Convert/UDINT/UDINT_TO_LREAL', node_UDINT_TO_LREAL);
NodeFactory.AddNodeAsPrototype('PLC/Convert/UDINT/UDINT_TO_REAL', node_UDINT_TO_REAL);

// flow 
NodeFactory.AddNodeAsPrototype('PLC/Flow/IF',nodeIf);
NodeFactory.AddNodeAsPrototype('PLC/Flow/IF_Merge', nodeIfMerge);
NodeFactory.AddNodeAsPrototype('PLC/Flow/For', nodeForNext);

// Logic
NodeFactory.AddNodeAsPrototype('PLC/Logic/NOT', node_NOT);
NodeFactory.AddNodeAsPrototype('PLC/Logic/AND', node_AND);
NodeFactory.AddNodeAsPrototype('PLC/Logic/NAND', node_NAND);
NodeFactory.AddNodeAsPrototype('PLC/Logic/OR', node_OR);
NodeFactory.AddNodeAsPrototype('PLC/Logic/NOR', node_NOR);
NodeFactory.AddNodeAsPrototype('PLC/Logic/XOR', node_XOR);
NodeFactory.AddNodeAsPrototype('PLC/Logic/XNOR', node_XNOR);

// Hardware
//NodeFactory.AddNodeAsPrototype('PLC/Hardware/DI', node_DigitalInput);
//NodeFactory.AddNodeAsPrototype('PLC/Hardware/DO', node_DigitalOutput);

// TwinCAT
//NodeFactory.AddNodeAsPrototype('PLC/TwinCAT/TwinCAT Status', node_TwinCATStatus);

// Strings
NodeFactory.AddNodeAsPrototype('PLC/Strings/CONCAT', node_CONCAT);
NodeFactory.AddNodeAsPrototype('PLC/Strings/DELETE', node_DELETE);
NodeFactory.AddNodeAsPrototype('PLC/Strings/FIND', node_FIND);
NodeFactory.AddNodeAsPrototype('PLC/Strings/INSERT', node_INSERT);
NodeFactory.AddNodeAsPrototype('PLC/Strings/LEFT', node_LEFT);
NodeFactory.AddNodeAsPrototype('PLC/Strings/LEN', node_LEN);
NodeFactory.AddNodeAsPrototype('PLC/Strings/MID', node_MID);
NodeFactory.AddNodeAsPrototype('PLC/Strings/REPLACE', node_REPLACE);
NodeFactory.AddNodeAsPrototype('PLC/Strings/RIGHT', node_RIGHT);

// Variable
//NodeFactory.AddNodeAsPrototype('PLC/Variable/SetByRef', node_SetByRef);
END_METHOD

END_FUNCTION_BLOCK

// ---- Nodes/TwinCAT/Node_TwinCATStatus.TcPOU
{attribute 'linkalways'} 
{attribute 'no_explicit_call' := 'This FB is a CLASS and must be accessed using methods or properties'}
{attribute 'enable_dynamic_creation'}
FUNCTION_BLOCK FINAL Node_TwinCATStatus EXTENDS Node
VAR
	lastPlcCycleTime : _ULINT(0);
	averagePlcCycleTime : _ULINT(0);
	usedMemory : _DWORD(0);
	avaliableMemory : _DWORD(0);
	maximumMemory : _DWORD(0);
	
	// node variables
	getRouterStatusInfo : FB_GetRouterStatusInfo;
	tcRouterStatusInfo : ST_TcRouterStatusInfo;
	cycleTimes : ARRAY [0..9] OF ULINT := [0,0,0,0,0,0,0,0,0,0];
    cycleTimeIndex : INT := 0;
END_VAR

METHOD PUBLIC  Clone : I_Node
VAR
	pNode : POINTER TO Node_TwinCATStatus;
END_VAR
pNode := __NEW(Node_TwinCATStatus);
Clone := pNode^;
END_METHOD

METHOD FB_init : BOOL
VAR_INPUT
	bInitRetains : BOOL; // if TRUE, the retain variables are initialized (warm start / cold start)
	bInCopyCode : BOOL;  // if TRUE, the instance afterwards gets moved into the copy code (online change)
END_VAR
AddContent('lastCycleTime', lastPlcCycleTime);
AddContent('averageCycleTime', averagePlcCycleTime);
AddContent('usedMemory', usedMemory);
AddContent('avaliableMemory', avaliableMemory);
AddContent('maximumMemory', maximumMemory);
END_METHOD

METHOD PROTECTED OnExecute
VAR
	i : INT;
    sum : ULINT := 0;
END_VAR
// memory 

IF NOT getRouterStatusInfo.bBusy THEN
	tcRouterStatusInfo := getRouterStatusInfo.info;
END_IF

getRouterStatusInfo(
	sNetId:= '' ,
	bExecute:= NOT getRouterStatusInfo.bBusy, 
	tTimeout:= T#5S, 
	bBusy=> , 
	bError=> , 
	nErrID=> , 
	info=> 
);

usedMemory.Value := tcRouterStatusInfo.maxMem - tcRouterStatusInfo.maxMemAvail;
avaliableMemory.Value := tcRouterStatusInfo.maxMemAvail;
maximumMemory.Value := tcRouterStatusInfo.maxMem;

// cycle time

cycleTimes[cycleTimeIndex] := F_GetTaskTotalTime(0);
cycleTimeIndex := (cycleTimeIndex + 1) MOD 10;

FOR i := 0 TO 9 DO
    sum := sum + cycleTimes[i];
END_FOR

lastPlcCycleTime.Value := F_GetTaskTotalTime(0);
averagePlcCycleTime.Value := sum / 10;
END_METHOD

END_FUNCTION_BLOCK

// ---- Nodes/Strings/Node_CONCAT.TcPOU
{attribute 'linkalways'} 
{attribute 'no_explicit_call' := 'This FB is a CLASS and must be accessed using methods or properties'}
{attribute 'enable_dynamic_creation'}
FUNCTION_BLOCK FINAL Node_CONCAT EXTENDS Node
VAR
	str1 : _STRING('');
    str2 : _STRING('');
	out : _STRING('');
END_VAR

METHOD PUBLIC  Clone : I_Node
VAR
	pNode : POINTER TO Node_CONCAT;
END_VAR
pNode := __NEW(Node_CONCAT);
Clone := pNode^;
END_METHOD

METHOD FB_init : BOOL
VAR_INPUT
	bInitRetains : BOOL; // if TRUE, the retain variables are initialized (warm start / cold start)
	bInCopyCode : BOOL;  // if TRUE, the instance afterwards gets moved into the copy code (online change)
END_VAR
AddParameter('str1', str1);
AddParameter('str2', str2);
AddOutput('out', out);
END_METHOD

METHOD PROTECTED OnExecute
VAR
END_VAR
out.Value := CONCAT(str1.Value, str2.Value);
END_METHOD

END_FUNCTION_BLOCK

// ---- Nodes/Strings/Node_DELETE.TcPOU
{attribute 'linkalways'} 
{attribute 'no_explicit_call' := 'This FB is a CLASS and must be accessed using methods or properties'}
{attribute 'enable_dynamic_creation'}
FUNCTION_BLOCK FINAL Node_DELETE EXTENDS Node
VAR
	str : _STRING('');
    len : _INT(0);
	pos : _INT(0);
	out : _STRING('');
END_VAR

METHOD PUBLIC  Clone : I_Node
VAR
	pNode : POINTER TO Node_DELETE;
END_VAR
pNode := __NEW(Node_DELETE);
Clone := pNode^;
END_METHOD

METHOD FB_init : BOOL
VAR_INPUT
	bInitRetains : BOOL; // if TRUE, the retain variables are initialized (warm start / cold start)
	bInCopyCode : BOOL;  // if TRUE, the instance afterwards gets moved into the copy code (online change)
END_VAR
AddParameter('str', str);
AddParameter('len', len);
AddParameter('pos', pos);
AddOutput('out', out);
END_METHOD

METHOD PROTECTED OnExecute
VAR
END_VAR
out.Value := DELETE(str.Value, len.Value, pos.Value);
END_METHOD

END_FUNCTION_BLOCK

// ---- Nodes/Strings/Node_FIND.TcPOU
{attribute 'linkalways'} 
{attribute 'no_explicit_call' := 'This FB is a CLASS and must be accessed using methods or properties'}
{attribute 'enable_dynamic_creation'}
FUNCTION_BLOCK FINAL Node_FIND EXTENDS Node
VAR
	str1 : _STRING('');
	str2 : _STRING('');
	out : _INT(0);
END_VAR

METHOD PUBLIC  Clone : I_Node
VAR
	pNode : POINTER TO Node_FIND;
END_VAR
pNode := __NEW(Node_FIND);
Clone := pNode^;
END_METHOD

METHOD FB_init : BOOL
VAR_INPUT
	bInitRetains : BOOL; // if TRUE, the retain variables are initialized (warm start / cold start)
	bInCopyCode : BOOL;  // if TRUE, the instance afterwards gets moved into the copy code (online change)
END_VAR
AddParameter('str1', str1);
AddParameter('str2', str2);
AddOutput('out', out);
END_METHOD

METHOD PROTECTED OnExecute
VAR
END_VAR
out.Value := FIND(str1.Value, str2.Value);
END_METHOD

END_FUNCTION_BLOCK

// ---- Nodes/Strings/Node_INSERT.TcPOU
{attribute 'linkalways'} 
{attribute 'no_explicit_call' := 'This FB is a CLASS and must be accessed using methods or properties'}
{attribute 'enable_dynamic_creation'}
FUNCTION_BLOCK FINAL Node_INSERT EXTENDS Node
VAR
	str1 : _STRING('');
    str2 : _STRING('');
	pos : _INT(0);
	out : _STRING('');
END_VAR

METHOD PUBLIC  Clone : I_Node
VAR
	pNode : POINTER TO Node_INSERT;
END_VAR
pNode := __NEW(Node_INSERT);
Clone := pNode^;
END_METHOD

METHOD FB_init : BOOL
VAR_INPUT
	bInitRetains : BOOL; // if TRUE, the retain variables are initialized (warm start / cold start)
	bInCopyCode : BOOL;  // if TRUE, the instance afterwards gets moved into the copy code (online change)
END_VAR
AddParameter('str1', str1);
AddParameter('str2', str2);
AddParameter('pos', pos);
AddOutput('out', out);
END_METHOD

METHOD PROTECTED OnExecute
VAR
END_VAR
out.Value := INSERT(str1.Value, str2.Value, pos.Value);
END_METHOD

END_FUNCTION_BLOCK

// ---- Nodes/Strings/Node_LEFT.TcPOU
{attribute 'linkalways'} 
{attribute 'no_explicit_call' := 'This FB is a CLASS and must be accessed using methods or properties'}
{attribute 'enable_dynamic_creation'}
FUNCTION_BLOCK FINAL Node_LEFT EXTENDS Node
VAR
	str : _STRING('');
	size : _INT(0);
	out : _STRING('');
END_VAR

METHOD PUBLIC  Clone : I_Node
VAR
	pNode : POINTER TO Node_LEFT;
END_VAR
pNode := __NEW(Node_LEFT);
Clone := pNode^;
END_METHOD

METHOD FB_init : BOOL
VAR_INPUT
	bInitRetains : BOOL; // if TRUE, the retain variables are initialized (warm start / cold start)
	bInCopyCode : BOOL;  // if TRUE, the instance afterwards gets moved into the copy code (online change)
END_VAR
AddParameter('str', str);
AddParameter('size', size);
AddOutput('out', out);
END_METHOD

METHOD PROTECTED OnExecute
VAR
END_VAR
out.Value := LEFT(str.Value, size.Value);
END_METHOD

END_FUNCTION_BLOCK

// ---- Nodes/Strings/Node_LEN.TcPOU
{attribute 'linkalways'} 
{attribute 'no_explicit_call' := 'This FB is a CLASS and must be accessed using methods or properties'}
{attribute 'enable_dynamic_creation'}
FUNCTION_BLOCK FINAL Node_LEN EXTENDS Node
VAR
	str : _STRING('');
	out : _INT(0);
END_VAR

METHOD PUBLIC  Clone : I_Node
VAR
	pNode : POINTER TO Node_LEN;
END_VAR
pNode := __NEW(Node_LEN);
Clone := pNode^;
END_METHOD

METHOD FB_init : BOOL
VAR_INPUT
	bInitRetains : BOOL; // if TRUE, the retain variables are initialized (warm start / cold start)
	bInCopyCode : BOOL;  // if TRUE, the instance afterwards gets moved into the copy code (online change)
END_VAR
AddParameter('str', str);
AddOutput('out', out);
END_METHOD

METHOD PROTECTED OnExecute
VAR
END_VAR
out.Value := LEN(str.Value);
END_METHOD

END_FUNCTION_BLOCK

// ---- Nodes/Strings/Node_MID.TcPOU
{attribute 'linkalways'} 
{attribute 'no_explicit_call' := 'This FB is a CLASS and must be accessed using methods or properties'}
{attribute 'enable_dynamic_creation'}
FUNCTION_BLOCK FINAL Node_MID EXTENDS Node
VAR
	str : _STRING('');
    len : _INT(0);
	pos : _INT(0);
	out : _STRING('');
END_VAR

METHOD PUBLIC  Clone : I_Node
VAR
	pNode : POINTER TO Node_MID;
END_VAR
pNode := __NEW(Node_MID);
Clone := pNode^;
END_METHOD

METHOD FB_init : BOOL
VAR_INPUT
	bInitRetains : BOOL; // if TRUE, the retain variables are initialized (warm start / cold start)
	bInCopyCode : BOOL;  // if TRUE, the instance afterwards gets moved into the copy code (online change)
END_VAR
AddParameter('str', str);
AddParameter('len', len);
AddParameter('pos', pos);
AddOutput('out', out);
END_METHOD

METHOD PROTECTED OnExecute
VAR
END_VAR
out.Value := MID(str.Value, len.Value, pos.Value);
END_METHOD

END_FUNCTION_BLOCK

// ---- Nodes/Strings/Node_REPLACE.TcPOU
{attribute 'linkalways'} 
{attribute 'no_explicit_call' := 'This FB is a CLASS and must be accessed using methods or properties'}
{attribute 'enable_dynamic_creation'}
FUNCTION_BLOCK FINAL Node_REPLACE EXTENDS Node
VAR
	str1 : _STRING('');
    str2 : _STRING('');
	l : _INT(0);
	p : _INT(0);
	out : _STRING('');
END_VAR

METHOD PUBLIC  Clone : I_Node
VAR
	pNode : POINTER TO Node_REPLACE;
END_VAR
pNode := __NEW(Node_REPLACE);
Clone := pNode^;
END_METHOD

METHOD FB_init : BOOL
VAR_INPUT
	bInitRetains : BOOL; // if TRUE, the retain variables are initialized (warm start / cold start)
	bInCopyCode : BOOL;  // if TRUE, the instance afterwards gets moved into the copy code (online change)
END_VAR
AddParameter('str1', str1);
AddParameter('str2', str2);
AddParameter('l', l);
AddParameter('p', p);
AddOutput('out', out);
END_METHOD

METHOD PROTECTED OnExecute
VAR
END_VAR
out.Value := REPLACE(str1.Value, str2.Value, l.Value, p.Value);
END_METHOD

END_FUNCTION_BLOCK

// ---- Nodes/Strings/Node_RIGHT.TcPOU
{attribute 'linkalways'} 
{attribute 'no_explicit_call' := 'This FB is a CLASS and must be accessed using methods or properties'}
{attribute 'enable_dynamic_creation'}
FUNCTION_BLOCK FINAL Node_RIGHT EXTENDS Node
VAR
	str : _STRING('');
	size : _INT(0);
	out : _STRING('');
END_VAR

METHOD PUBLIC  Clone : I_Node
VAR
	pNode : POINTER TO Node_RIGHT;
END_VAR
pNode := __NEW(Node_RIGHT);
Clone := pNode^;
END_METHOD

METHOD FB_init : BOOL
VAR_INPUT
	bInitRetains : BOOL; // if TRUE, the retain variables are initialized (warm start / cold start)
	bInCopyCode : BOOL;  // if TRUE, the instance afterwards gets moved into the copy code (online change)
END_VAR
AddParameter('str', str);
AddParameter('size', size);
AddOutput('out', out);
END_METHOD

METHOD PROTECTED OnExecute
VAR
END_VAR
out.Value := RIGHT(str.Value, size.Value);
END_METHOD

END_FUNCTION_BLOCK

// ---- Nodes/Variable/Node_SetByRef.TcPOU
{attribute 'linkalways'} 
{attribute 'no_explicit_call' := 'This FB is a CLASS and must be accessed using methods or properties'}
{attribute 'enable_dynamic_creation'}
FUNCTION_BLOCK Node_SetByRef EXTENDS Node
VAR
	byRef : _ANY();
	value : _ANY();
END_VAR

METHOD PUBLIC  Clone : I_Node
VAR_INPUT
END_VAR
VAR
	pNode : POINTER TO Node_SetByRef;
END_VAR
pNode := __NEW(Node_SetByRef);
Clone := pNode^;
END_METHOD

METHOD FB_init : BOOL
VAR_INPUT
	bInitRetains : BOOL; // if TRUE, the retain variables are initialized (warm start / cold start)
	bInCopyCode : BOOL;  // if TRUE, the instance afterwards gets moved into the copy code (online change)
END_VAR
AddInputWithGroup('byRef', byRef, 'T');
AddInputWithGroup('value', value, 'T');
AddOutputWithGroup('byRef', byRef, 'T');
END_METHOD

METHOD PROTECTED  OnExecute
byRef.TryCopyFrom(value);
END_METHOD

END_FUNCTION_BLOCK

// ---- PlcPack.TcPOU
{attribute 'linkalways'} 
{attribute 'no_explicit_call' := 'This FB is a CLASS and must be accessed using methods or properties'}
{attribute 'enable_dynamic_creation'}
FUNCTION_BLOCK PlcPack IMPLEMENTS I_GraphPack
VAR
	plcDatatypePack : PlcDatatypePack;
	plcNodePack : PlcNodePack;
END_VAR

METHOD Register
VAR_INPUT
	Datatypes : I_Datatypes;
	NodeFactory : I_NodeFactory;
END_VAR
plcDatatypePack.RegisterWithDatatypes(Datatypes);
plcNodePack.RegisterWithNodeFactory(NodeFactory);
END_METHOD

END_FUNCTION_BLOCK
